{region '#Template'}
	{attribute 'Category' := 'Universal'}
	{attribute 'Version' := '0.0.1.0'}
	{attribute 'Tags' := 'Universal, Motor, Aggregate'}
	{attribute 'Description' := 'Motor 1 stufig	// Motor 1 stage'}
{endregion}
FUNCTION_BLOCK FB_BA_Mot1st EXTENDS FB_BA_AggregateB
VAR_OUTPUT
	bCmd		: BOOL;
END_VAR
VAR_INPUT CONSTANT
	Dst			: FB_BA_BI_IO;
	
	Cmd			: FB_BA_BO_IO;							
END_VAR

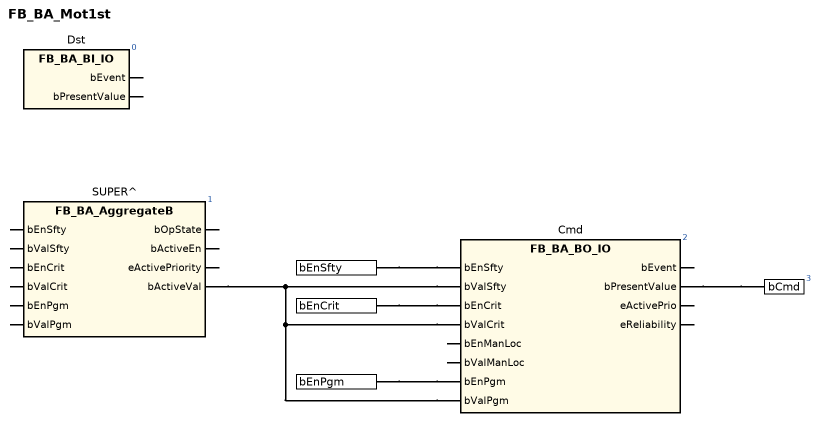
Dst(); // FB_BA_BI_IO
SUPER^(); // FB_BA_AggregateB
Cmd(
    bEnSfty := bEnSfty,
    bValSfty := SUPER^.bActiveVal,
    bEnCrit := bEnCrit,
    bValCrit := SUPER^.bActiveVal,
    bEnPgm := bEnPgm,
    bValPgm := SUPER^.bActiveVal); // FB_BA_BO_IO
bCmd := Cmd.bPresentValue;

METHOD FB_init : BOOL
VAR_INPUT
	bInitRetains : BOOL; // if TRUE, the retain variables are initialized (warm start / cold start)
	bInCopyCode : BOOL;  // if TRUE, the instance afterwards gets moved into the copy code (online change)
END_VAR
Dst.iParent							:= THIS^;
Dst.iLabel							:= LblUniFieldDevice.Motor_Dst;	
Dst.sObjectName						:= '{Idx=01}';	
Dst.sDeviceType						:= '';
Dst.bEnOutOfService					:= FALSE;
Dst.ePolarity						:= E_BA_Polarity.eReverse;
Dst.sActiveText 					:= Texts.txtTriggered;
Dst.sInactiveText 					:= Texts.txtNormal;
Dst.nStateChangeCount				:= 0;
Dst.nActiveTimeElapsed				:= 0;
Dst.nEventClassID					:= EventClasses.AlarmTechnicalExtended;
Dst.stTimeDelay.nToNormal			:= BA2_Param.nDefTimeDelay_ToNormal;
Dst.stTimeDelay.nToAbnormal			:= BA2_Param.nDefTimeDelay_ToAbnormal;
Dst.bAlarmValue						:= TRUE;
Dst.bAcknowledgeRm					:= FALSE;	
Dst.aEventTransitionText[1]			:= Texts.txtTriggered;
Dst.aEventTransitionText[2]			:= Texts.txtError;
Dst.aEventTransitionText[3]			:= Texts.txtNormal;
Dst.bEventDetectionEnable			:= TRUE;
Dst.eEnPlantLock					:= E_BA_LockPriority.eLocalMedium;

Cmd.iParent							:= THIS^;
Cmd.iLabel							:= LblUniFieldDevice.Motor_Cmd;			
Cmd.sObjectName						:= '{Idx=01}';
Cmd.sDeviceType						:= '';	
Cmd.ePolarity						:= E_BA_Polarity.eNormal;
Cmd.eFeedbackPolarity				:= E_BA_Polarity.eNormal;
Cmd.eOverriddenPolarity				:= E_BA_Polarity.eReverse;
Cmd.sActiveText 					:= Texts.txtOn;
Cmd.sInactiveText 					:= Texts.txtOff;
Cmd.nStateChangeCount				:= 0;
Cmd.nActiveTimeElapsed				:= 0;
Cmd.nMinimumOnTime					:= 0;
Cmd.nMinimumOffTime					:= 0;
Cmd.bEnManualRm						:= FALSE;	//	Priority  8	
Cmd.bValManualRm					:= FALSE;	//	Priority  8
Cmd.bDefaultValue					:= FALSE;
Cmd.nEventClassID					:= EventClasses.DisturbanceExtended;
Cmd.stTimeDelay.nToNormal			:= BA2_Param.nDefTimeDelay_ToNormal;
Cmd.stTimeDelay.nToAbnormal			:= BA2_Param.nDefTimeDelay_ToAbnormal;
Cmd.bAcknowledgeRm					:= FALSE;		
Cmd.aEventTransitionText[1]			:= Texts.txtDisturb;
Cmd.aEventTransitionText[2]			:= Texts.txtNone;
Cmd.aEventTransitionText[3]			:= Texts.txtNormal;
Cmd.bEventDetectionEnable			:= FALSE;
Cmd.eEnPlantLock					:= E_BA_LockPriority.eNoLock;
END_METHOD

END_FUNCTION_BLOCK

(* stored: Version 1.1.0.1, ProductVersion 3.1.4024.6
   POU FB_BA_Mot1st: Id {72abe04b-ec04-4b91-85fb-f82e8a153f11}, SpecialFunc None
   Method FB_init: Id {84aadd14-79a7-483b-bbd6-49ce4093678f} *)
